// TIA Portal V18 export
// export: Created 2025-12-01T17:53:13.674237Z, ExportSetting None, DisplayName Totally Integrated Automation Portal, DisplayVersion V18 Update 5, DisplayName TIA Portal Openness, DisplayVersion V18 Update 5, DisplayName TIA Portal Teamcenter Gateway, DisplayVersion V18, DisplayName TIA Portal Version Control Interface, DisplayVersion V18, DisplayName STEP 7 Professional, DisplayVersion V18 Update 5, DisplayName STEP 7 Safety, DisplayVersion V18, DisplayName WinCC Professional, DisplayVersion V18 Update 5
Screen "820 User"  1280x800, Number=820, Template=08CtrlPanel
  ScreenLayer "Layer_0"
    UserView "用户视图_1"  Appearance=Appearance3D, StyleItem=Benutzeranzeige
    Button "btnMenu5_1" at 384,725 size 128x75  Authorization=User administration, StyleItem=BtnActive20, TextOff="用户设定 / User Config / Užívateľ Konfigurácia"
      on Click: ActivateScreen(Screen name := , Object number := 0); SetTag(Tag := Sys_VersionManagement_HMIPageID, Value := 820)
